// TIA Portal V17 export
// export: Created 2026-04-13T11:12:42.173199Z, ExportSetting WithDefaults, DisplayName Totally Integrated Automation Portal, DisplayVersion V17 Update 4, DisplayName TIA Portal Openness, DisplayVersion V17 Update 4, DisplayName TIA Portal Version Control Interface, DisplayVersion V17, DisplayName SINAMICS Startdrive Advanced, DisplayVersion V17, DisplayName SINAMICS Startdrive G130, G150, S120, S150, SINAMICS MV, S210, DisplayVersion V17, DisplayName SINAMICS Startdrive G110M, G120, G120C, G120D, G120P, G115D, DisplayVersion V17, DisplayName STEP 7 Professional, DisplayVersion V17 Update 4, DisplayName STEP 7 Safety, DisplayVersion V17, DisplayName WinCC Professional, DisplayVersion V17 Update 4
FUNCTION_BLOCK "步段延迟案例"   // FB70, SCL
{ S7_Optimized_Access := 'TRUE' }
VERSION : 0.1
// stored: AutoNumber true, IsIECCheckEnabled false, IsRetainMemResEnabled false, MemoryReserve 100, SetENOAutomatically false, UDAEnableTagReadback false
   VAR_IN_OUT
      BD步段运行 : Int;
      BD步段设定 : Int;
   END_VAR
   VAR
      STEP1 { S7_SetPoint := 'True'} : "步段延迟";
      STEP2 { S7_SetPoint := 'True'} : "步段延迟";
      STEP3 { S7_SetPoint := 'True'} : "步段延迟";
   END_VAR
BEGIN
   CASE #BD步段运行 OF
       1:
           #STEP1.AND := #BD步段运行 = 1;
           #STEP1(YC延迟设定时间:=30.0);


           IF #STEP1.Q THEN
               #BD步段运行 := 2;
           END_IF;
           ;
       2:
           #STEP2.AND := #BD步段运行 = 2;
           #STEP2(YC延迟设定时间 := 30.0);
           IF #STEP2.Q THEN


               #BD步段运行 := 3;
           END_IF;
           ;
       3:
           #STEP3.AND := #BD步段运行 = 3;
           #STEP3(YC延迟设定时间 := 30.0);
           IF #STEP3.Q THEN
               #BD步段运行 := 1;
           END_IF;

   END_CASE;


   IF #BD步段设定 <> #BD步段运行 THEN
       #STEP1.YX运行时间 := 0;
       #STEP2.YX运行时间 := 0;
       #STEP3.YX运行时间 := 0;
       #STEP1.Q := 0;
       #STEP2.Q := 0;
       #STEP3.Q := 0;
       #BD步段设定 := #BD步段运行;
   END_IF;
END_FUNCTION_BLOCK
